FUNCTION fMeanFilter : REAL
VAR_INPUT
	rInputValue:REAL;
	rDelta:REAL;
END_VAR
VAR_IN_OUT
	rMeanValue:REAL;
END_VAR
VAR
END_VAR

rDelta := LIMIT(1,rDelta,100);
IF ABS(0.20*rMeanValue) < ABS( (rMeanValue - rInputValue)/rDelta) THEN
	rMeanValue := rInputValue;
END_IF
rMeanValue := rMeanValue - (rMeanValue - rInputValue)/rDelta;

END_FUNCTION

(* stored: Version 1.1.0.1, ProductVersion 3.1.4024.15
   POU fMeanFilter: Id {31274a27-acb0-4bbe-8c53-61018b8909fd}, SpecialFunc None *)
